FUNCTION_BLOCK FB_SOLVEALFABETA
VAR_INPUT
x : REAL;
y : REAL;
END_VAR
VAR_OUTPUT
alfa : REAL;
beta : REAL;
d1 : REAL;
d2 : REAL;
alfa1 : REAL;
alfa2 : REAL;
beta1 : REAL;
beta2 : REAL;
error: BOOL := 0;

END_VAR
VAR
END_VAR

error:=FALSE;
d1 := SQRT(y*y+(x+GVL.d)*(x+GVL.d));
IF d1>(GVL.l1*GVL.l1+GVL.l2*GVL.l2) THEN
	error:=TRUE;
END_IF
d2 := SQRT(y*y+(x-GVL.d)*(x-GVL.d));
IF d2>(GVL.l1*GVL.l1+GVL.l2*GVL.l2) THEN
	error:=TRUE;
END_IF

alfa1 := ATAN (y/(x+GVL.d));
IF alfa1 < 0 THEN
	error:=TRUE;
END_IF
beta1 := GVL.Pi	+ ATAN (y/(x-GVL.d));
IF beta1 < 0 THEN
	error:=TRUE;
END_IF

IF (ABS((GVL.l1*GVL.l1+d1*d1-GVL.l2*GVL.l2)/(2*GVL.l1*d1))>1) THEN
error := TRUE;
END_IF

IF (ABS((GVL.l1*GVL.l1+d2*d2-GVL.l2*GVL.l2)/(2*GVL.l1*d2))>1) THEN
error := TRUE;
END_IF

IF error=FALSE THEN
	alfa2 := ABS(ACOS((GVL.l1*GVL.l1+d1*d1-GVL.l2*GVL.l2)/(2*GVL.l1*d1)));
	beta2 := ABS(ACOS((GVL.l1*GVL.l1+d2*d2-GVL.l2*GVL.l2)/(2*GVL.l1*d2)));
alfa := alfa1 + alfa2;
beta := beta1 - beta2;

END_IF

END_FUNCTION_BLOCK

(* stored: Version 1.1.0.1, ProductVersion 3.1.4024.4
   POU FB_SOLVEALFABETA: Id {fa1b62a0-c717-4454-9065-b5fc8a73063a}, SpecialFunc None *)
